// Mitsubishi GX Works2 project: project   PLC: Q03UDV

PROGRAM MAIN
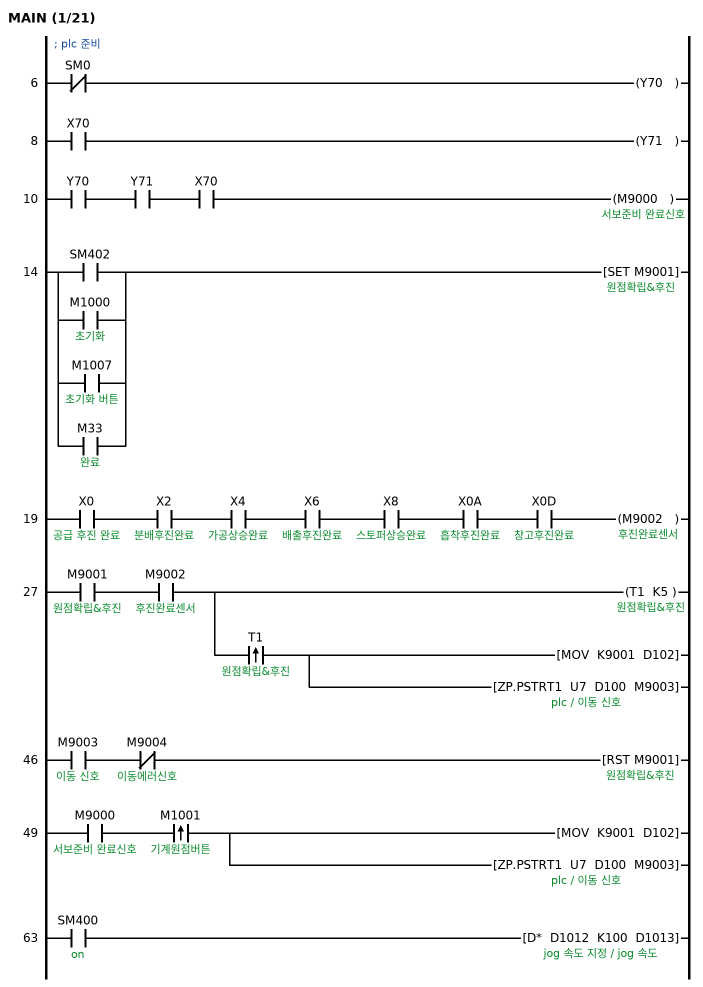
; plc 준비
6     LDI     SM0
      OUT     Y70
8     LD      X70
      OUT     Y71
10    LD      Y70
      AND     Y71
      AND     X70
      OUT     M9000  ; 서보준비 완료신호
14    LD      SM402
      OR      M1000  ; 초기화
      OR      M1007  ; 초기화 버튼
      OR      M33  ; 완료
      SET     M9001  ; 원점확립&후진
19    LD      X0  ; 공급 후진 완료
      AND     X2  ; 분배후진완료
      AND     X4  ; 가공상승완료
      AND     X6  ; 배출후진완료
      AND     X8  ; 스토퍼상승완료
      AND     X0A  ; 흡착후진완료
      AND     X0D  ; 창고후진완료
      OUT     M9002  ; 후진완료센서
27    LD      M9001  ; 원점확립&후진
      AND     M9002  ; 후진완료센서
      OUT     T1 K5  ; 원점확립&후진
      ANDP    T1  ; 원점확립&후진
      MOV     K9001 D102
      ZP.PSTRT1 U7 D100 M9003  ; plc / 이동 신호
46    LD      M9003  ; 이동 신호
      ANI     M9004  ; 이동에러신호
      RST     M9001  ; 원점확립&후진
49    LD      M9000  ; 서보준비 완료신호
      ANDP    M1001  ; 기계원점버튼
      MOV     K9001 D102
      ZP.PSTRT1 U7 D100 M9003
63    LD      SM400  ; on
      D*      D1012 K100 D1013  ; jog 속도 지정 / jog 속도
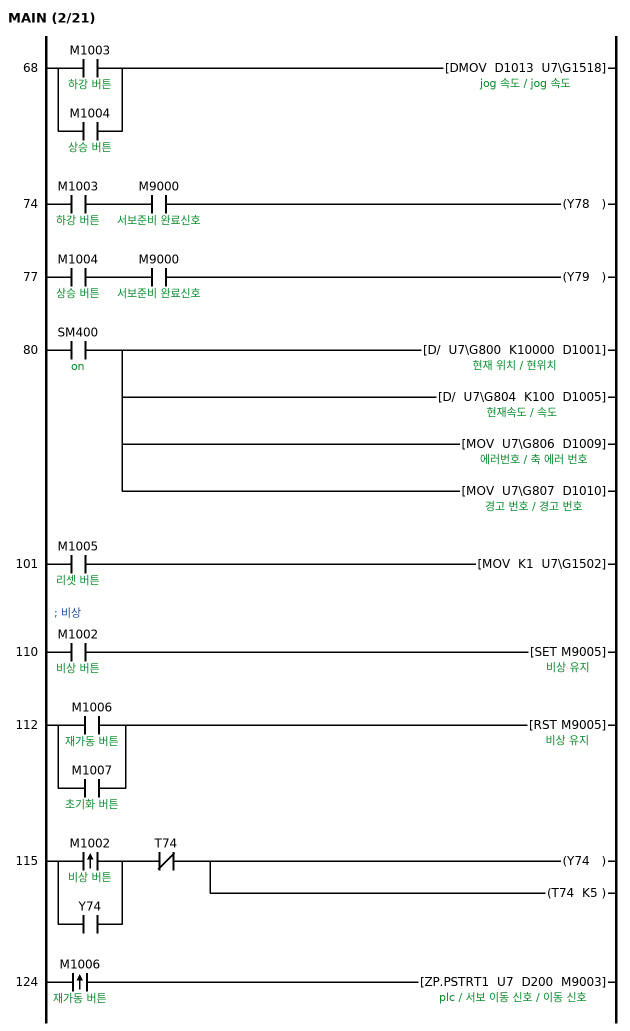
68    LD      M1003  ; 하강 버튼
      OR      M1004  ; 상승 버튼
      DMOV    D1013 U7\G1518  ; jog 속도
74    LD      M1003  ; 하강 버튼
      AND     M9000  ; 서보준비 완료신호
      OUT     Y78
77    LD      M1004  ; 상승 버튼
      AND     M9000  ; 서보준비 완료신호
      OUT     Y79
80    LD      SM400  ; on
      D/      U7\G800 K10000 D1001  ; 현재 위치 / 현위치
      D/      U7\G804 K100 D1005  ; 현재속도 / 속도
      MOV     U7\G806 D1009  ; 에러번호 / 축 에러 번호
      MOV     U7\G807 D1010  ; 경고 번호 / 경고 번호
101   LD      M1005  ; 리셋 버튼
      MOV     K1 U7\G1502
; 비상
110   LD      M1002  ; 비상 버튼
      SET     M9005  ; 비상 유지
112   LD      M1006  ; 재가동 버튼
      OR      M1007  ; 초기화 버튼
      RST     M9005  ; 비상 유지
115   LDP     M1002  ; 비상 버튼
      OR      Y74
      ANI     T74
      OUT     Y74
      OUT     T74 K5
124   LDP     M1006  ; 재가동 버튼
      ZP.PSTRT1 U7 D200 M9003  ; 서보 이동 신호
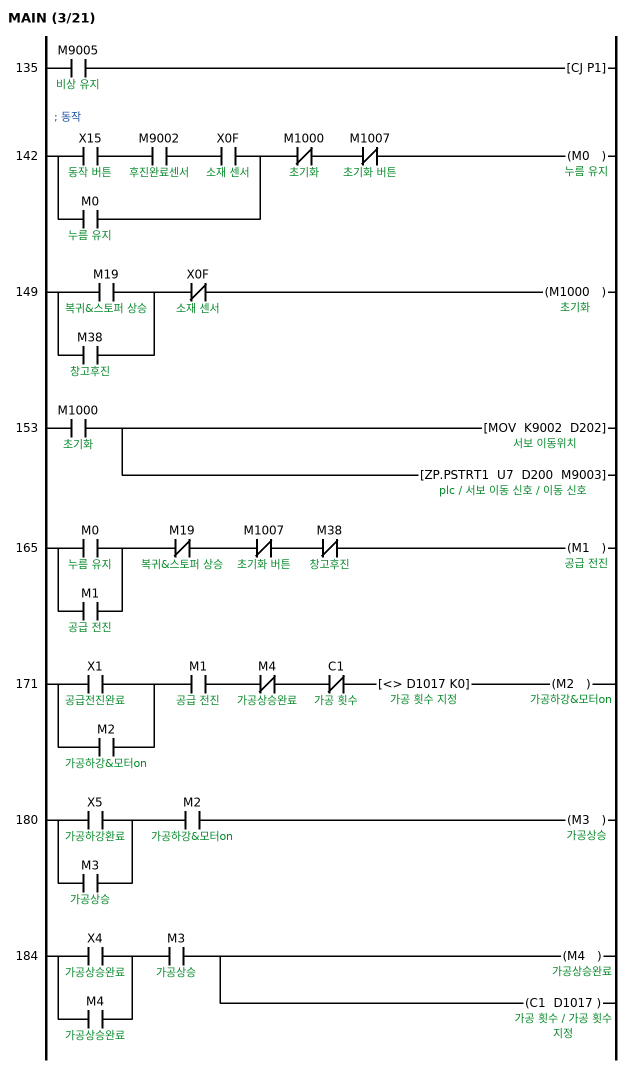
135   LD      M9005  ; 비상 유지
      CJ      P1  ; 비상
; 동작
142   LD      X15  ; 동작 버튼
      AND     M9002  ; 후진완료센서
      AND     X0F  ; 소재 센서
      OR      M0  ; 누름 유지
      ANI     M1000  ; 초기화
      ANI     M1007  ; 초기화 버튼
      OUT     M0  ; 누름 유지
149   LD      M19  ; 복귀&스토퍼 상승
      OR      M38  ; 창고후진
      ANI     X0F  ; 소재 센서
      OUT     M1000  ; 초기화
153   LD      M1000  ; 초기화
      MOV     K9002 D202  ; 서보 이동위치
      ZP.PSTRT1 U7 D200 M9003
165   LD      M0  ; 누름 유지
      OR      M1  ; 공급 전진
      ANI     M19  ; 복귀&스토퍼 상승
      ANI     M1007  ; 초기화 버튼
      ANI     M38  ; 창고후진
      OUT     M1  ; 공급 전진
171   LD      X1  ; 공급전진완료
      OR      M2  ; 가공하강&모터on
      AND     M1  ; 공급 전진
      ANI     M4  ; 가공상승완료
      ANI     C1  ; 가공 횟수
      AND<>   D1017 K0  ; 가공 횟수 지정
      OUT     M2  ; 가공하강&모터on
180   LD      X5  ; 가공하강환료
      OR      M3  ; 가공상승
      AND     M2  ; 가공하강&모터on
      OUT     M3  ; 가공상승
184   LD      X4  ; 가공상승완료
      OR      M4  ; 가공상승완료
      AND     M3  ; 가공상승
      OUT     M4  ; 가공상승완료
      OUT     C1 D1017  ; 가공 횟수 / 가공 횟수 지정
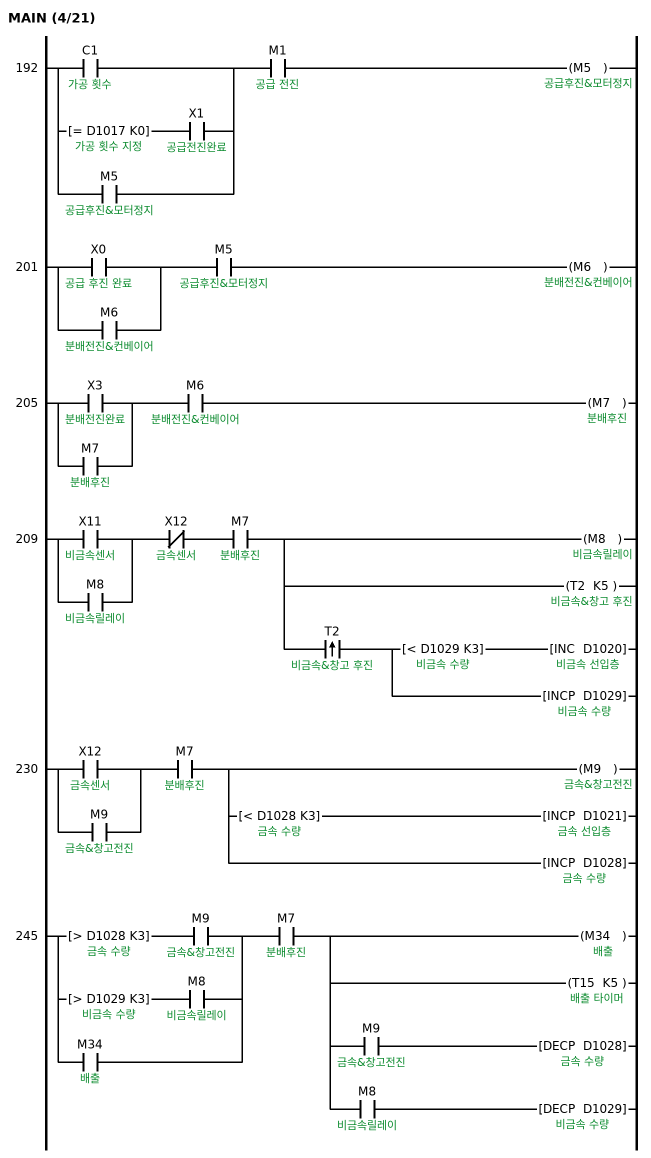
192   LD      C1  ; 가공 횟수
      LD=     D1017 K0  ; 가공 횟수 지정
      AND     X1  ; 공급전진완료
      ORB
      OR      M5  ; 공급후진&모터정지
      AND     M1  ; 공급 전진
      OUT     M5  ; 공급후진&모터정지
201   LD      X0  ; 공급 후진 완료
      OR      M6  ; 분배전진&컨베이어
      AND     M5  ; 공급후진&모터정지
      OUT     M6  ; 분배전진&컨베이어
205   LD      X3  ; 분배전진완료
      OR      M7  ; 분배후진
      AND     M6  ; 분배전진&컨베이어
      OUT     M7  ; 분배후진
209   LD      X11  ; 비금속센서
      OR      M8  ; 비금속릴레이
      ANI     X12  ; 금속센서
      AND     M7  ; 분배후진
      OUT     M8  ; 비금속릴레이
      OUT     T2 K5  ; 비금속&창고 후진
      ANDP    T2  ; 비금속&창고 후진
      MPS
      AND<    D1029 K3  ; 비금속 수량
      INC     D1020  ; 비금속 선입층
      MPP
      INCP    D1029
230   LD      X12  ; 금속센서
      OR      M9  ; 금속&창고전진
      AND     M7  ; 분배후진
      OUT     M9  ; 금속&창고전진
      MPS
      AND<    D1028 K3  ; 금속 수량
      INCP    D1021  ; 금속 선입층
      MPP
      INCP    D1028
245   LD>     D1028 K3  ; 금속 수량
      AND     M9  ; 금속&창고전진
      LD>     D1029 K3  ; 비금속 수량
      AND     M8  ; 비금속릴레이
      ORB
      OR      M34  ; 배출
      AND     M7  ; 분배후진
      OUT     M34  ; 배출
      OUT     T15 K5  ; 배출 타이머
      MPS
      AND     M9  ; 금속&창고전진
      DECP    D1028
      MPP
      AND     M8  ; 비금속릴레이
      DECP    D1029
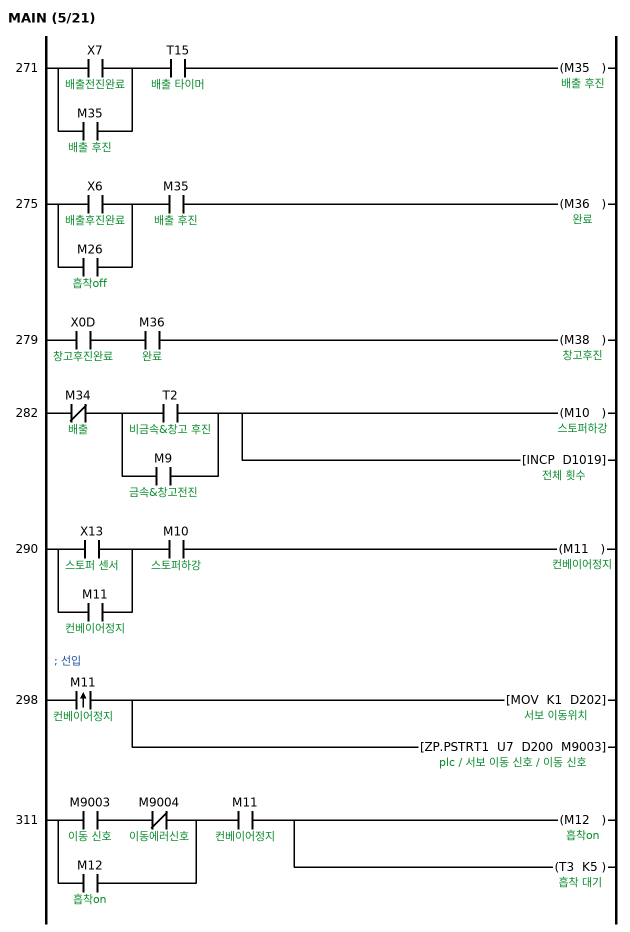
271   LD      X7  ; 배출전진완료
      OR      M35  ; 배출 후진
      AND     T15  ; 배출 타이머
      OUT     M35  ; 배출 후진
275   LD      X6  ; 배출후진완료
      OR      M26  ; 흡착off
      AND     M35  ; 배출 후진
      OUT     M36  ; 완료
279   LD      X0D  ; 창고후진완료
      AND     M36  ; 완료
      OUT     M38  ; 창고후진
282   LDI     M34  ; 배출
      LD      T2  ; 비금속&창고 후진
      OR      M9  ; 금속&창고전진
      ANB
      OUT     M10  ; 스토퍼하강
      INCP    D1019  ; 전체 횟수
290   LD      X13  ; 스토퍼 센서
      OR      M11  ; 컨베이어정지
      AND     M10  ; 스토퍼하강
      OUT     M11  ; 컨베이어정지
; 선입
298   LDP     M11  ; 컨베이어정지
      MOV     K1 D202
      ZP.PSTRT1 U7 D200 M9003
311   LD      M9003  ; 이동 신호
      ANI     M9004  ; 이동에러신호
      OR      M12  ; 흡착on
      AND     M11  ; 컨베이어정지
      OUT     M12  ; 흡착on
      OUT     T3 K5  ; 흡착 대기
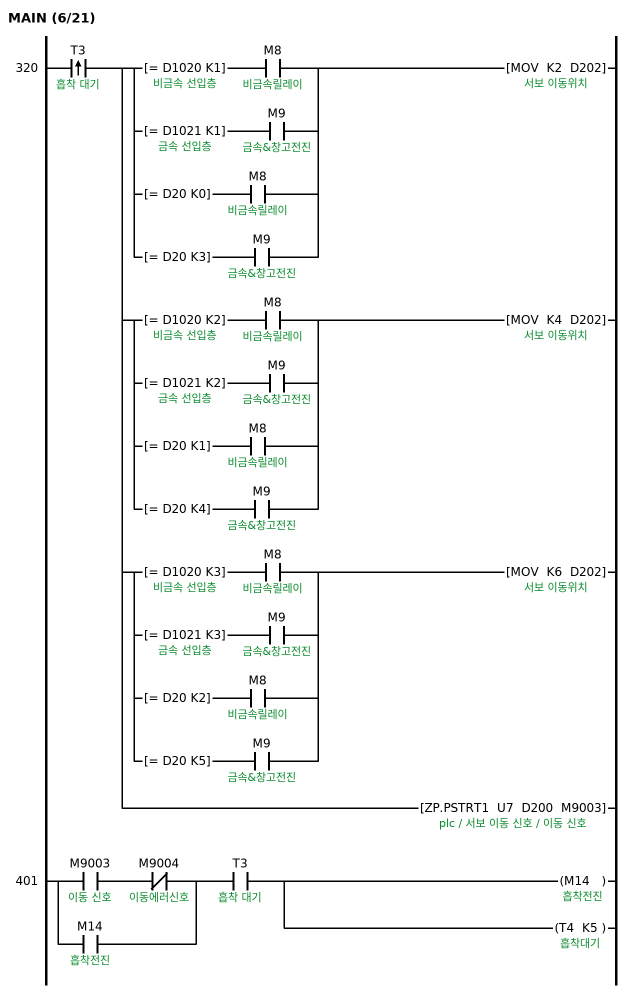
320   LDP     T3  ; 흡착 대기
      MPS
      LD=     D1020 K1  ; 비금속 선입층
      AND     M8  ; 비금속릴레이
      LD=     D1021 K1  ; 금속 선입층
      AND     M9  ; 금속&창고전진
      ORB
      LD=     D20 K0
      AND     M8  ; 비금속릴레이
      ORB
      LD=     D20 K3
      AND     M9  ; 금속&창고전진
      ORB
      ANB
      MOV     K2 D202
      MRD
      LD=     D1020 K2  ; 비금속 선입층
      AND     M8  ; 비금속릴레이
      LD=     D1021 K2  ; 금속 선입층
      AND     M9  ; 금속&창고전진
      ORB
      LD=     D20 K1
      AND     M8  ; 비금속릴레이
      ORB
      LD=     D20 K4
      AND     M9  ; 금속&창고전진
      ORB
      ANB
      MOV     K4 D202
      MRD
      LD=     D1020 K3  ; 비금속 선입층
      AND     M8  ; 비금속릴레이
      LD=     D1021 K3  ; 금속 선입층
      AND     M9  ; 금속&창고전진
      ORB
      LD=     D20 K2
      AND     M8  ; 비금속릴레이
      ORB
      LD=     D20 K5
      AND     M9  ; 금속&창고전진
      ORB
      ANB
      MOV     K6 D202
      MPP
      ZP.PSTRT1 U7 D200 M9003
401   LD      M9003  ; 이동 신호
      ANI     M9004  ; 이동에러신호
      OR      M14  ; 흡착전진
      AND     T3  ; 흡착 대기
      OUT     M14  ; 흡착전진
      OUT     T4 K5  ; 흡착대기
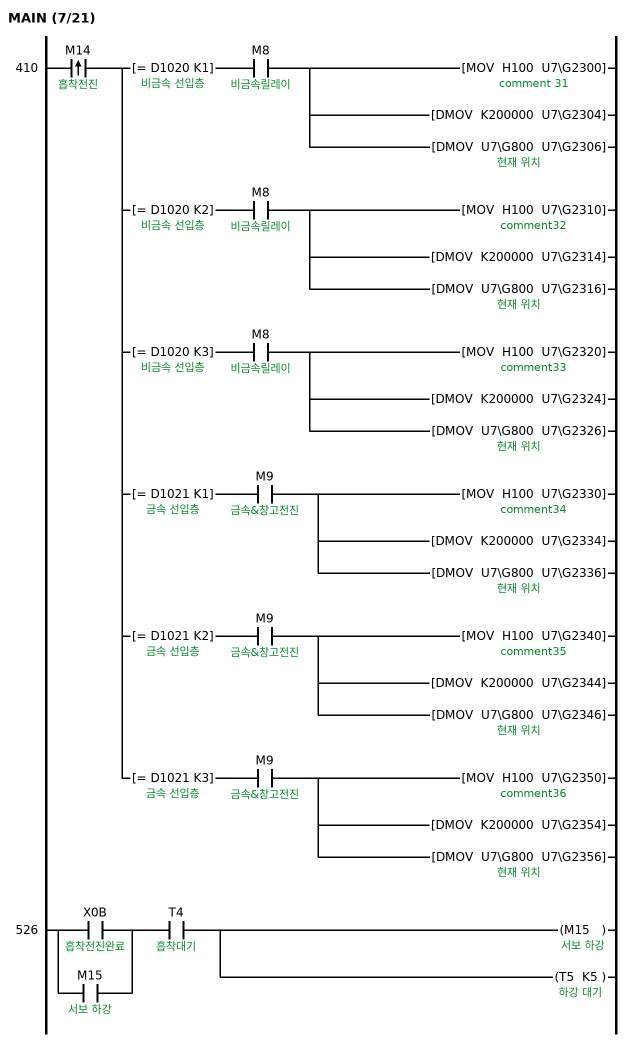
410   LDP     M14  ; 흡착전진
      MPS
      AND=    D1020 K1  ; 비금속 선입층
      AND     M8  ; 비금속릴레이
      MOV     H100 U7\G2300  ; comment 31
      DMOV    K200000 U7\G2304
      DMOV    U7\G800 U7\G2306
      MRD
      AND=    D1020 K2  ; 비금속 선입층
      AND     M8  ; 비금속릴레이
      MOV     H100 U7\G2310  ; comment32
      DMOV    K200000 U7\G2314
      DMOV    U7\G800 U7\G2316
      MRD
      AND=    D1020 K3  ; 비금속 선입층
      AND     M8  ; 비금속릴레이
      MOV     H100 U7\G2320  ; comment33
      DMOV    K200000 U7\G2324
      DMOV    U7\G800 U7\G2326
      MRD
      AND=    D1021 K1  ; 금속 선입층
      AND     M9  ; 금속&창고전진
      MOV     H100 U7\G2330  ; comment34
      DMOV    K200000 U7\G2334
      DMOV    U7\G800 U7\G2336
      MRD
      AND=    D1021 K2  ; 금속 선입층
      AND     M9  ; 금속&창고전진
      MOV     H100 U7\G2340  ; comment35
      DMOV    K200000 U7\G2344
      DMOV    U7\G800 U7\G2346
      MPP
      AND=    D1021 K3  ; 금속 선입층
      AND     M9  ; 금속&창고전진
      MOV     H100 U7\G2350  ; comment36
      DMOV    K200000 U7\G2354
      DMOV    U7\G800 U7\G2356
526   LD      X0B  ; 흡착전진완료
      OR      M15  ; 서보 하강
      AND     T4  ; 흡착대기
      OUT     M15  ; 서보 하강
      OUT     T5 K5  ; 하강 대기
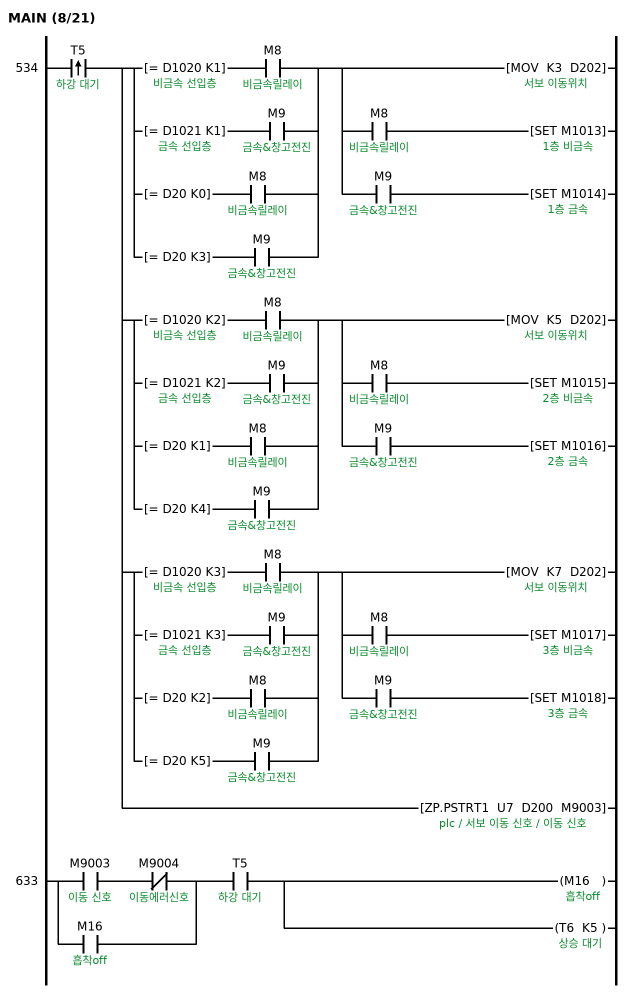
534   LDP     T5  ; 하강 대기
      MPS
      LD=     D1020 K1  ; 비금속 선입층
      AND     M8  ; 비금속릴레이
      LD=     D1021 K1  ; 금속 선입층
      AND     M9  ; 금속&창고전진
      ORB
      LD=     D20 K0
      AND     M8  ; 비금속릴레이
      ORB
      LD=     D20 K3
      AND     M9  ; 금속&창고전진
      ORB
      ANB
      MOV     K3 D202
      MPS
      AND     M8  ; 비금속릴레이
      SET     M1013  ; 1층 비금속
      MPP
      AND     M9  ; 금속&창고전진
      SET     M1014  ; 1층 금속
      MRD
      LD=     D1020 K2  ; 비금속 선입층
      AND     M8  ; 비금속릴레이
      LD=     D1021 K2  ; 금속 선입층
      AND     M9  ; 금속&창고전진
      ORB
      LD=     D20 K1
      AND     M8  ; 비금속릴레이
      ORB
      LD=     D20 K4
      AND     M9  ; 금속&창고전진
      ORB
      ANB
      MOV     K5 D202
      MPS
      AND     M8  ; 비금속릴레이
      SET     M1015  ; 2층 비금속
      MPP
      AND     M9  ; 금속&창고전진
      SET     M1016  ; 2층 금속
      MRD
      LD=     D1020 K3  ; 비금속 선입층
      AND     M8  ; 비금속릴레이
      LD=     D1021 K3  ; 금속 선입층
      AND     M9  ; 금속&창고전진
      ORB
      LD=     D20 K2
      AND     M8  ; 비금속릴레이
      ORB
      LD=     D20 K5
      AND     M9  ; 금속&창고전진
      ORB
      ANB
      MOV     K7 D202
      MPS
      AND     M8  ; 비금속릴레이
      SET     M1017  ; 3층 비금속
      MPP
      AND     M9  ; 금속&창고전진
      SET     M1018  ; 3층 금속
      MPP
      ZP.PSTRT1 U7 D200 M9003
633   LD      M9003  ; 이동 신호
      ANI     M9004  ; 이동에러신호
      OR      M16  ; 흡착off
      AND     T5  ; 하강 대기
      OUT     M16  ; 흡착off
      OUT     T6 K5  ; 상승 대기
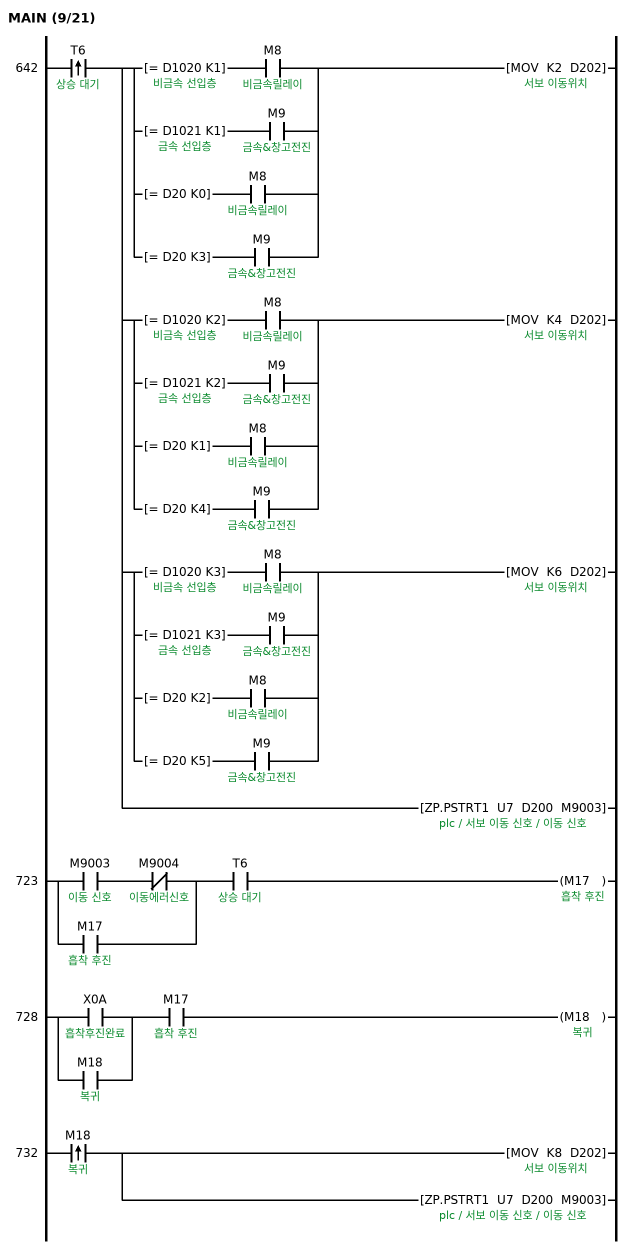
642   LDP     T6  ; 상승 대기
      MPS
      LD=     D1020 K1  ; 비금속 선입층
      AND     M8  ; 비금속릴레이
      LD=     D1021 K1  ; 금속 선입층
      AND     M9  ; 금속&창고전진
      ORB
      LD=     D20 K0
      AND     M8  ; 비금속릴레이
      ORB
      LD=     D20 K3
      AND     M9  ; 금속&창고전진
      ORB
      ANB
      MOV     K2 D202
      MRD
      LD=     D1020 K2  ; 비금속 선입층
      AND     M8  ; 비금속릴레이
      LD=     D1021 K2  ; 금속 선입층
      AND     M9  ; 금속&창고전진
      ORB
      LD=     D20 K1
      AND     M8  ; 비금속릴레이
      ORB
      LD=     D20 K4
      AND     M9  ; 금속&창고전진
      ORB
      ANB
      MOV     K4 D202
      MRD
      LD=     D1020 K3  ; 비금속 선입층
      AND     M8  ; 비금속릴레이
      LD=     D1021 K3  ; 금속 선입층
      AND     M9  ; 금속&창고전진
      ORB
      LD=     D20 K2
      AND     M8  ; 비금속릴레이
      ORB
      LD=     D20 K5
      AND     M9  ; 금속&창고전진
      ORB
      ANB
      MOV     K6 D202
      MPP
      ZP.PSTRT1 U7 D200 M9003
723   LD      M9003  ; 이동 신호
      ANI     M9004  ; 이동에러신호
      OR      M17  ; 흡착 후진
      AND     T6  ; 상승 대기
      OUT     M17  ; 흡착 후진
728   LD      X0A  ; 흡착후진완료
      OR      M18  ; 복귀
      AND     M17  ; 흡착 후진
      OUT     M18  ; 복귀
732   LDP     M18  ; 복귀
      MOV     K8 D202
      ZP.PSTRT1 U7 D200 M9003
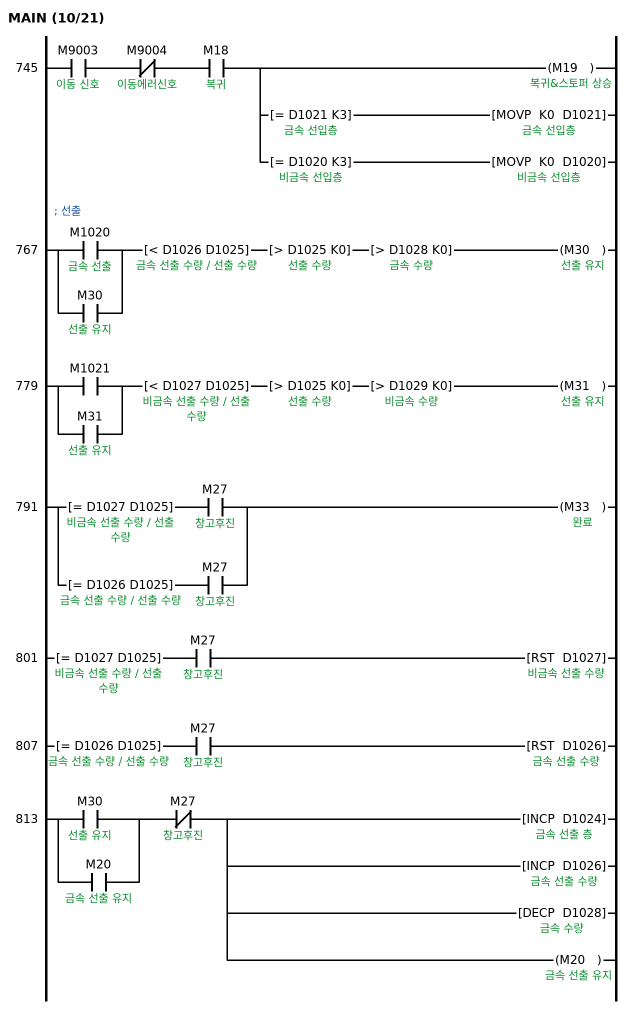
745   LD      M9003  ; 이동 신호
      ANI     M9004  ; 이동에러신호
      AND     M18  ; 복귀
      OUT     M19  ; 복귀&스토퍼 상승
      MPS
      AND=    D1021 K3  ; 금속 선입층
      MOVP    K0 D1021
      MPP
      AND=    D1020 K3  ; 비금속 선입층
      MOVP    K0 D1020
; 선출
767   LD      M1020  ; 금속 선출
      OR      M30  ; 선출 유지
      AND<    D1026 D1025  ; 금속 선출 수량 / 선출 수량
      AND>    D1025 K0  ; 선출 수량
      AND>    D1028 K0  ; 금속 수량
      OUT     M30  ; 선출 유지
779   LD      M1021
      OR      M31  ; 선출 유지
      AND<    D1027 D1025  ; 비금속 선출 수량 / 선출 수량
      AND>    D1025 K0  ; 선출 수량
      AND>    D1029 K0  ; 비금속 수량
      OUT     M31  ; 선출 유지
791   LD=     D1027 D1025  ; 비금속 선출 수량 / 선출 수량
      AND     M27  ; 창고후진
      LD=     D1026 D1025  ; 금속 선출 수량 / 선출 수량
      AND     M27  ; 창고후진
      ORB
      OUT     M33  ; 완료
801   LD=     D1027 D1025  ; 비금속 선출 수량 / 선출 수량
      AND     M27  ; 창고후진
      RST     D1027  ; 비금속 선출 수량
807   LD=     D1026 D1025  ; 금속 선출 수량 / 선출 수량
      AND     M27  ; 창고후진
      RST     D1026  ; 금속 선출 수량
813   LD      M30  ; 선출 유지
      OR      M20  ; 금속 선출 유지
      ANI     M27  ; 창고후진
      INCP    D1024  ; 금속 선출 층
      INCP    D1026
      DECP    D1028
      OUT     M20  ; 금속 선출 유지
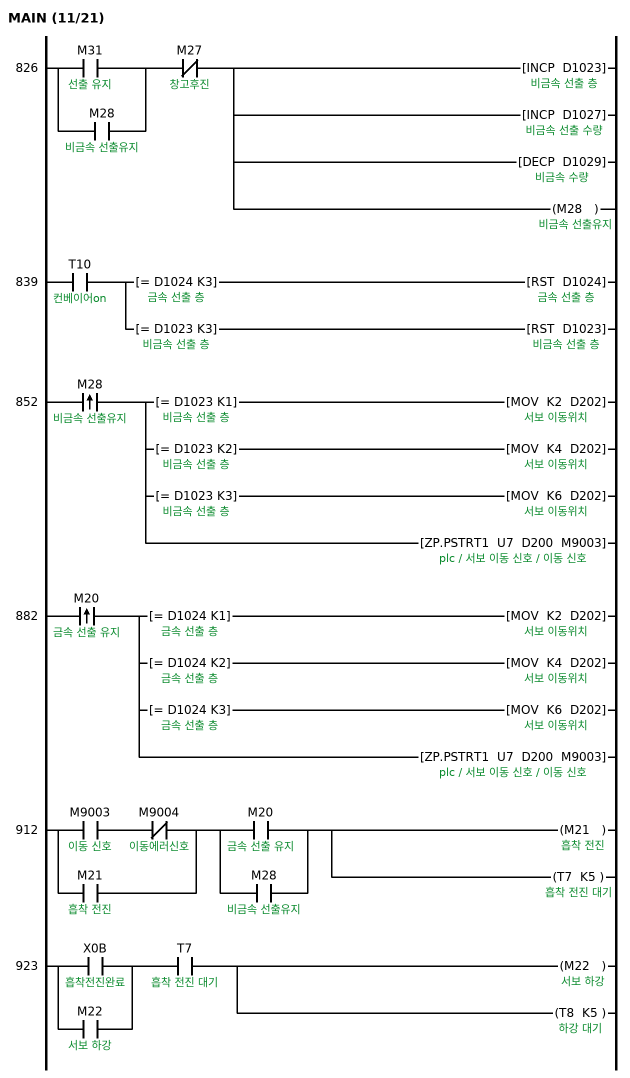
826   LD      M31  ; 선출 유지
      OR      M28  ; 비금속 선출유지
      ANI     M27  ; 창고후진
      INCP    D1023  ; 비금속 선출 층
      INCP    D1027
      DECP    D1029
      OUT     M28  ; 비금속 선출유지
839   LD      T10  ; 컨베이어on
      MPS
      AND=    D1024 K3  ; 금속 선출 층
      RST     D1024  ; 금속 선출 층
      MPP
      AND=    D1023 K3  ; 비금속 선출 층
      RST     D1023  ; 비금속 선출 층
852   LDP     M28  ; 비금속 선출유지
      MPS
      AND=    D1023 K1  ; 비금속 선출 층
      MOV     K2 D202
      MRD
      AND=    D1023 K2  ; 비금속 선출 층
      MOV     K4 D202
      MRD
      AND=    D1023 K3  ; 비금속 선출 층
      MOV     K6 D202
      MPP
      ZP.PSTRT1 U7 D200 M9003
882   LDP     M20  ; 금속 선출 유지
      MPS
      AND=    D1024 K1  ; 금속 선출 층
      MOV     K2 D202
      MRD
      AND=    D1024 K2  ; 금속 선출 층
      MOV     K4 D202
      MRD
      AND=    D1024 K3  ; 금속 선출 층
      MOV     K6 D202
      MPP
      ZP.PSTRT1 U7 D200 M9003
912   LD      M9003  ; 이동 신호
      ANI     M9004  ; 이동에러신호
      OR      M21  ; 흡착 전진
      LD      M20  ; 금속 선출 유지
      OR      M28  ; 비금속 선출유지
      ANB
      OUT     M21  ; 흡착 전진
      OUT     T7 K5  ; 흡착 전진 대기
923   LD      X0B  ; 흡착전진완료
      OR      M22  ; 서보 하강
      AND     T7  ; 흡착 전진 대기
      OUT     M22  ; 서보 하강
      OUT     T8 K5  ; 하강 대기
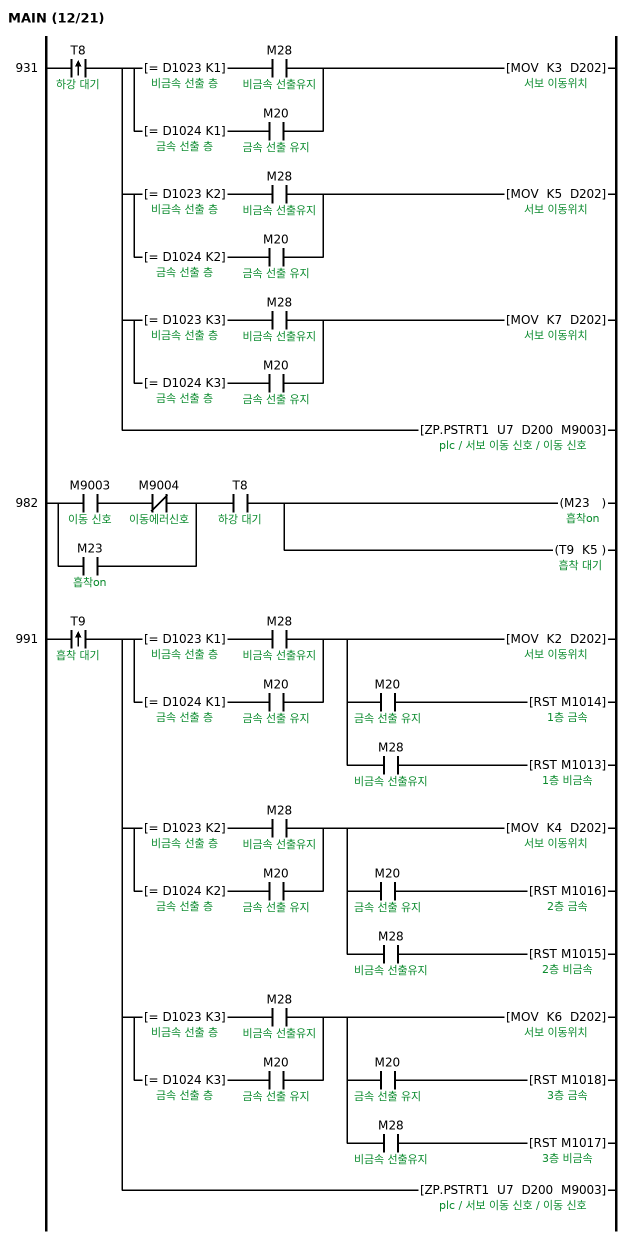
931   LDP     T8  ; 하강 대기
      MPS
      LD=     D1023 K1  ; 비금속 선출 층
      AND     M28  ; 비금속 선출유지
      LD=     D1024 K1  ; 금속 선출 층
      AND     M20  ; 금속 선출 유지
      ORB
      ANB
      MOV     K3 D202
      MRD
      LD=     D1023 K2  ; 비금속 선출 층
      AND     M28  ; 비금속 선출유지
      LD=     D1024 K2  ; 금속 선출 층
      AND     M20  ; 금속 선출 유지
      ORB
      ANB
      MOV     K5 D202
      MRD
      LD=     D1023 K3  ; 비금속 선출 층
      AND     M28  ; 비금속 선출유지
      LD=     D1024 K3  ; 금속 선출 층
      AND     M20  ; 금속 선출 유지
      ORB
      ANB
      MOV     K7 D202
      MPP
      ZP.PSTRT1 U7 D200 M9003
982   LD      M9003  ; 이동 신호
      ANI     M9004  ; 이동에러신호
      OR      M23  ; 흡착on
      AND     T8  ; 하강 대기
      OUT     M23  ; 흡착on
      OUT     T9 K5  ; 흡착 대기
991   LDP     T9  ; 흡착 대기
      MPS
      LD=     D1023 K1  ; 비금속 선출 층
      AND     M28  ; 비금속 선출유지
      LD=     D1024 K1  ; 금속 선출 층
      AND     M20  ; 금속 선출 유지
      ORB
      ANB
      MOV     K2 D202
      MPS
      AND     M20  ; 금속 선출 유지
      RST     M1014  ; 1층 금속
      MPP
      AND     M28  ; 비금속 선출유지
      RST     M1013  ; 1층 비금속
      MRD
      LD=     D1023 K2  ; 비금속 선출 층
      AND     M28  ; 비금속 선출유지
      LD=     D1024 K2  ; 금속 선출 층
      AND     M20  ; 금속 선출 유지
      ORB
      ANB
      MOV     K4 D202
      MPS
      AND     M20  ; 금속 선출 유지
      RST     M1016  ; 2층 금속
      MPP
      AND     M28  ; 비금속 선출유지
      RST     M1015  ; 2층 비금속
      MRD
      LD=     D1023 K3  ; 비금속 선출 층
      AND     M28  ; 비금속 선출유지
      LD=     D1024 K3  ; 금속 선출 층
      AND     M20  ; 금속 선출 유지
      ORB
      ANB
      MOV     K6 D202
      MPS
      AND     M20  ; 금속 선출 유지
      RST     M1018  ; 3층 금속
      MPP
      AND     M28  ; 비금속 선출유지
      RST     M1017  ; 3층 비금속
      MPP
      ZP.PSTRT1 U7 D200 M9003
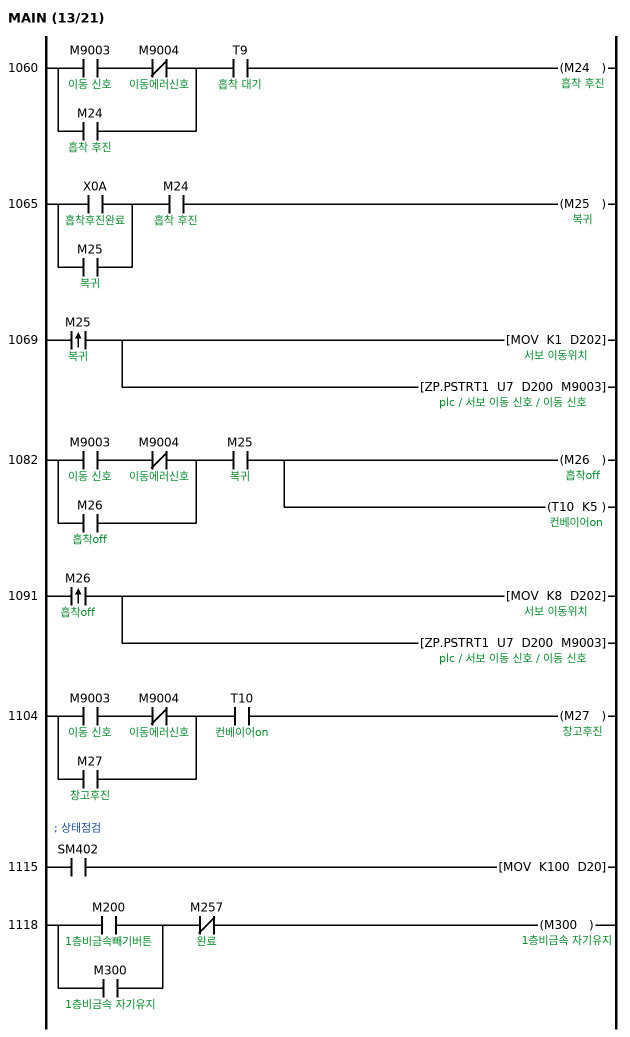
1060  LD      M9003  ; 이동 신호
      ANI     M9004  ; 이동에러신호
      OR      M24  ; 흡착 후진
      AND     T9  ; 흡착 대기
      OUT     M24  ; 흡착 후진
1065  LD      X0A  ; 흡착후진완료
      OR      M25  ; 복귀
      AND     M24  ; 흡착 후진
      OUT     M25  ; 복귀
1069  LDP     M25  ; 복귀
      MOV     K1 D202
      ZP.PSTRT1 U7 D200 M9003
1082  LD      M9003  ; 이동 신호
      ANI     M9004  ; 이동에러신호
      OR      M26  ; 흡착off
      AND     M25  ; 복귀
      OUT     M26  ; 흡착off
      OUT     T10 K5  ; 컨베이어on
1091  LDP     M26  ; 흡착off
      MOV     K8 D202
      ZP.PSTRT1 U7 D200 M9003
1104  LD      M9003  ; 이동 신호
      ANI     M9004  ; 이동에러신호
      OR      M27  ; 창고후진
      AND     T10  ; 컨베이어on
      OUT     M27  ; 창고후진
; 상태점검
1115  LD      SM402
      MOV     K100 D20
1118  LD      M200  ; 1층비금속빼기버튼
      OR      M300  ; 1층비금속 자기유지
      ANI     M257  ; 완료
      OUT     M300  ; 1층비금속 자기유지
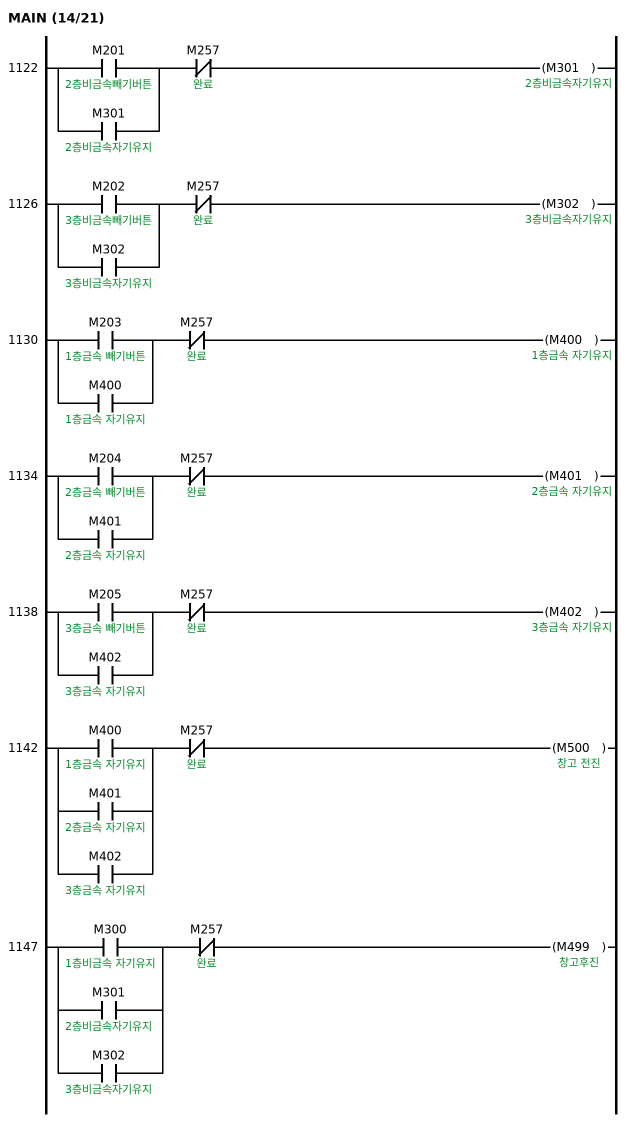
1122  LD      M201  ; 2층비금속빼기버튼
      OR      M301  ; 2층비금속자기유지
      ANI     M257  ; 완료
      OUT     M301  ; 2층비금속자기유지
1126  LD      M202  ; 3층비금속빼기버튼
      OR      M302  ; 3층비금속자기유지
      ANI     M257  ; 완료
      OUT     M302  ; 3층비금속자기유지
1130  LD      M203  ; 1층금속 빼기버튼
      OR      M400  ; 1층금속 자기유지
      ANI     M257  ; 완료
      OUT     M400  ; 1층금속 자기유지
1134  LD      M204  ; 2층금속 빼기버튼
      OR      M401  ; 2층금속 자기유지
      ANI     M257  ; 완료
      OUT     M401  ; 2층금속 자기유지
1138  LD      M205  ; 3층금속 빼기버튼
      OR      M402  ; 3층금속 자기유지
      ANI     M257  ; 완료
      OUT     M402  ; 3층금속 자기유지
1142  LD      M400  ; 1층금속 자기유지
      OR      M401  ; 2층금속 자기유지
      OR      M402  ; 3층금속 자기유지
      ANI     M257  ; 완료
      OUT     M500  ; 창고 전진
1147  LD      M300  ; 1층비금속 자기유지
      OR      M301  ; 2층비금속자기유지
      OR      M302  ; 3층비금속자기유지
      ANI     M257  ; 완료
      OUT     M499  ; 창고후진
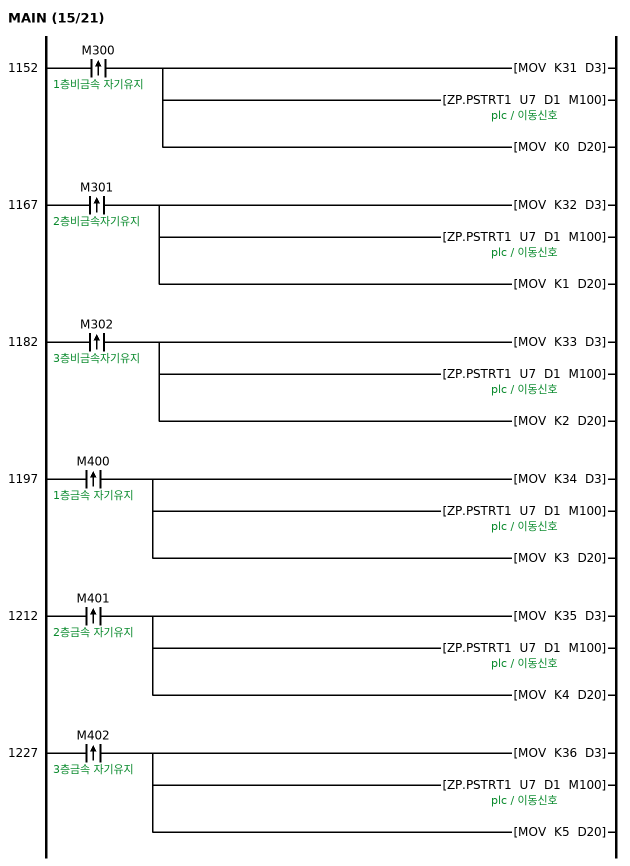
1152  LDP     M300  ; 1층비금속 자기유지
      MOV     K31 D3
      ZP.PSTRT1 U7 D1 M100  ; 이동신호
      MOV     K0 D20
1167  LDP     M301  ; 2층비금속자기유지
      MOV     K32 D3
      ZP.PSTRT1 U7 D1 M100
      MOV     K1 D20
1182  LDP     M302  ; 3층비금속자기유지
      MOV     K33 D3
      ZP.PSTRT1 U7 D1 M100
      MOV     K2 D20
1197  LDP     M400  ; 1층금속 자기유지
      MOV     K34 D3
      ZP.PSTRT1 U7 D1 M100
      MOV     K3 D20
1212  LDP     M401  ; 2층금속 자기유지
      MOV     K35 D3
      ZP.PSTRT1 U7 D1 M100
      MOV     K4 D20
1227  LDP     M402  ; 3층금속 자기유지
      MOV     K36 D3
      ZP.PSTRT1 U7 D1 M100
      MOV     K5 D20
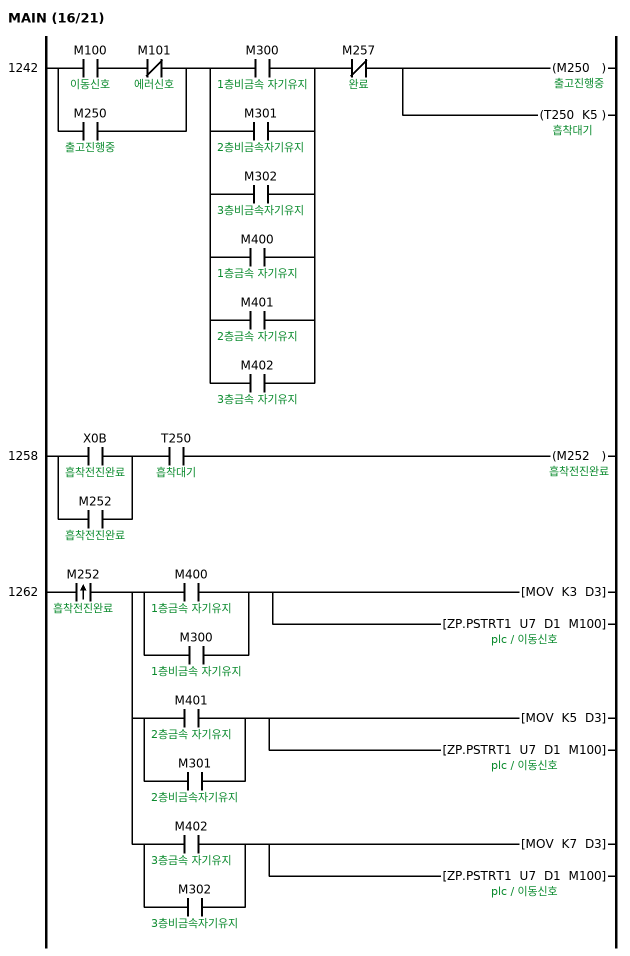
1242  LD      M100  ; 이동신호
      ANI     M101  ; 에러신호
      OR      M250  ; 출고진행중
      LD      M300  ; 1층비금속 자기유지
      OR      M301  ; 2층비금속자기유지
      OR      M302  ; 3층비금속자기유지
      OR      M400  ; 1층금속 자기유지
      OR      M401  ; 2층금속 자기유지
      OR      M402  ; 3층금속 자기유지
      ANB
      ANI     M257  ; 완료
      OUT     M250  ; 출고진행중
      OUT     T250 K5  ; 흡착대기
1258  LD      X0B  ; 흡착전진완료
      OR      M252  ; 흡착전진완료
      AND     T250  ; 흡착대기
      OUT     M252  ; 흡착전진완료
1262  LDP     M252  ; 흡착전진완료
      MPS
      LD      M400  ; 1층금속 자기유지
      OR      M300  ; 1층비금속 자기유지
      ANB
      MOV     K3 D3
      ZP.PSTRT1 U7 D1 M100
      MRD
      LD      M401  ; 2층금속 자기유지
      OR      M301  ; 2층비금속자기유지
      ANB
      MOV     K5 D3
      ZP.PSTRT1 U7 D1 M100
      MPP
      LD      M402  ; 3층금속 자기유지
      OR      M302  ; 3층비금속자기유지
      ANB
      MOV     K7 D3
      ZP.PSTRT1 U7 D1 M100
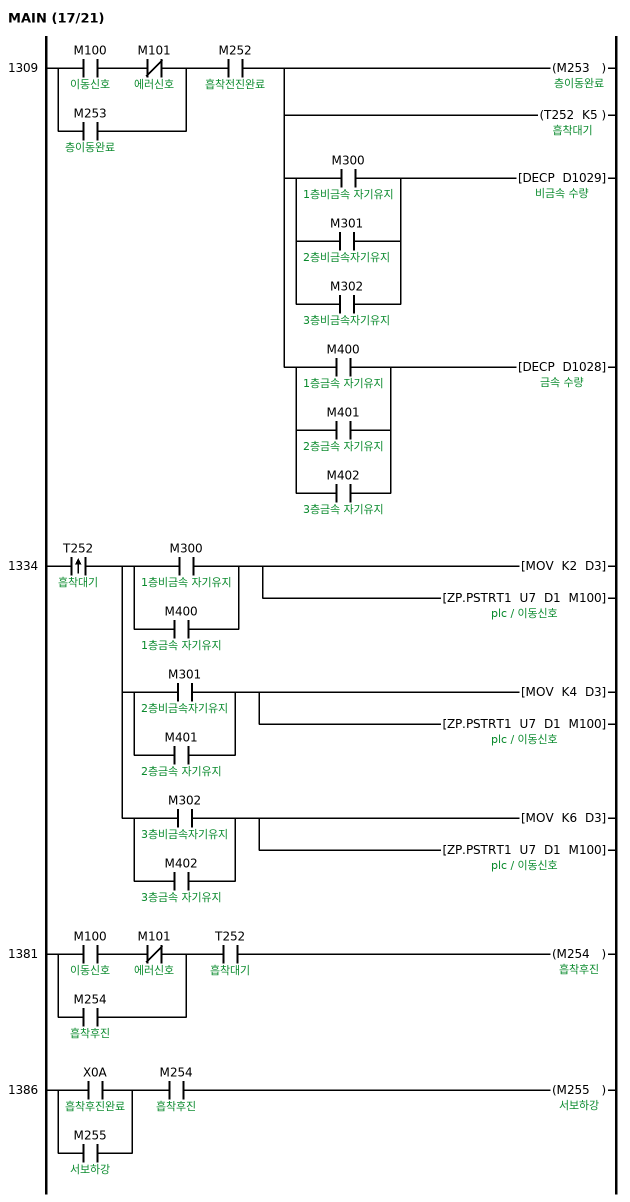
1309  LD      M100  ; 이동신호
      ANI     M101  ; 에러신호
      OR      M253  ; 층이동완료
      AND     M252  ; 흡착전진완료
      OUT     M253  ; 층이동완료
      OUT     T252 K5  ; 흡착대기
      MPS
      LD      M300  ; 1층비금속 자기유지
      OR      M301  ; 2층비금속자기유지
      OR      M302  ; 3층비금속자기유지
      ANB
      DECP    D1029
      MPP
      LD      M400  ; 1층금속 자기유지
      OR      M401  ; 2층금속 자기유지
      OR      M402  ; 3층금속 자기유지
      ANB
      DECP    D1028
1334  LDP     T252  ; 흡착대기
      MPS
      LD      M300  ; 1층비금속 자기유지
      OR      M400  ; 1층금속 자기유지
      ANB
      MOV     K2 D3
      ZP.PSTRT1 U7 D1 M100
      MRD
      LD      M301  ; 2층비금속자기유지
      OR      M401  ; 2층금속 자기유지
      ANB
      MOV     K4 D3
      ZP.PSTRT1 U7 D1 M100
      MPP
      LD      M302  ; 3층비금속자기유지
      OR      M402  ; 3층금속 자기유지
      ANB
      MOV     K6 D3
      ZP.PSTRT1 U7 D1 M100
1381  LD      M100  ; 이동신호
      ANI     M101  ; 에러신호
      OR      M254  ; 흡착후진
      AND     T252  ; 흡착대기
      OUT     M254  ; 흡착후진
1386  LD      X0A  ; 흡착후진완료
      OR      M255  ; 서보하강
      AND     M254  ; 흡착후진
      OUT     M255  ; 서보하강
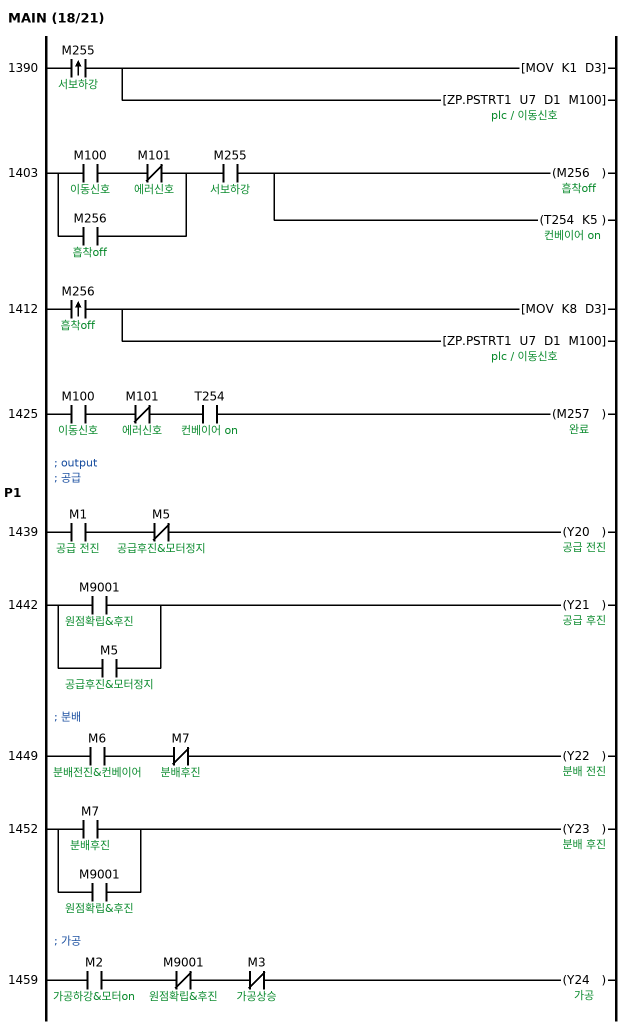
1390  LDP     M255  ; 서보하강
      MOV     K1 D3
      ZP.PSTRT1 U7 D1 M100
1403  LD      M100  ; 이동신호
      ANI     M101  ; 에러신호
      OR      M256  ; 흡착off
      AND     M255  ; 서보하강
      OUT     M256  ; 흡착off
      OUT     T254 K5  ; 컨베이어 on
1412  LDP     M256  ; 흡착off
      MOV     K8 D3
      ZP.PSTRT1 U7 D1 M100
1425  LD      M100  ; 이동신호
      ANI     M101  ; 에러신호
      AND     T254  ; 컨베이어 on
      OUT     M257  ; 완료
; output
; 공급
      P1
1439  LD      M1  ; 공급 전진
      ANI     M5  ; 공급후진&모터정지
      OUT     Y20  ; 공급 전진
1442  LD      M9001  ; 원점확립&후진
      OR      M5  ; 공급후진&모터정지
      OUT     Y21  ; 공급 후진
; 분배
1449  LD      M6  ; 분배전진&컨베이어
      ANI     M7  ; 분배후진
      OUT     Y22  ; 분배 전진
1452  LD      M7  ; 분배후진
      OR      M9001  ; 원점확립&후진
      OUT     Y23  ; 분배 후진
; 가공
1459  LD      M2  ; 가공하강&모터on
      ANI     M9001  ; 원점확립&후진
      ANI     M3  ; 가공상승
      OUT     Y24  ; 가공
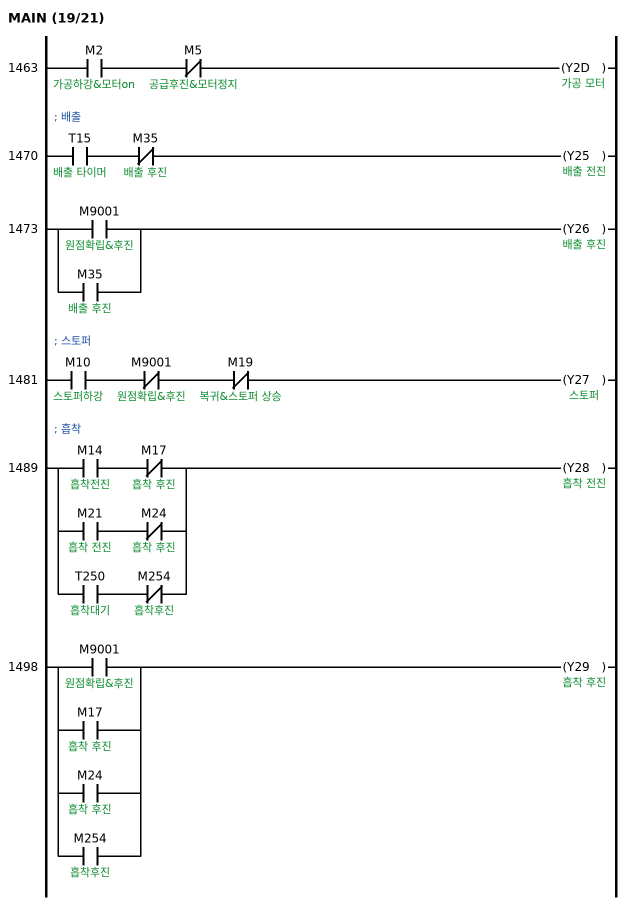
1463  LD      M2  ; 가공하강&모터on
      ANI     M5  ; 공급후진&모터정지
      OUT     Y2D  ; 가공 모터
; 배출
1470  LD      T15  ; 배출 타이머
      ANI     M35  ; 배출 후진
      OUT     Y25  ; 배출 전진
1473  LD      M9001  ; 원점확립&후진
      OR      M35  ; 배출 후진
      OUT     Y26  ; 배출 후진
; 스토퍼
1481  LD      M10  ; 스토퍼하강
      ANI     M9001  ; 원점확립&후진
      ANI     M19  ; 복귀&스토퍼 상승
      OUT     Y27  ; 스토퍼
; 흡착
1489  LD      M14  ; 흡착전진
      ANI     M17  ; 흡착 후진
      LD      M21  ; 흡착 전진
      ANI     M24  ; 흡착 후진
      ORB
      LD      T250  ; 흡착대기
      ANI     M254  ; 흡착후진
      ORB
      OUT     Y28  ; 흡착 전진
1498  LD      M9001  ; 원점확립&후진
      OR      M17  ; 흡착 후진
      OR      M24  ; 흡착 후진
      OR      M254  ; 흡착후진
      OUT     Y29  ; 흡착 후진
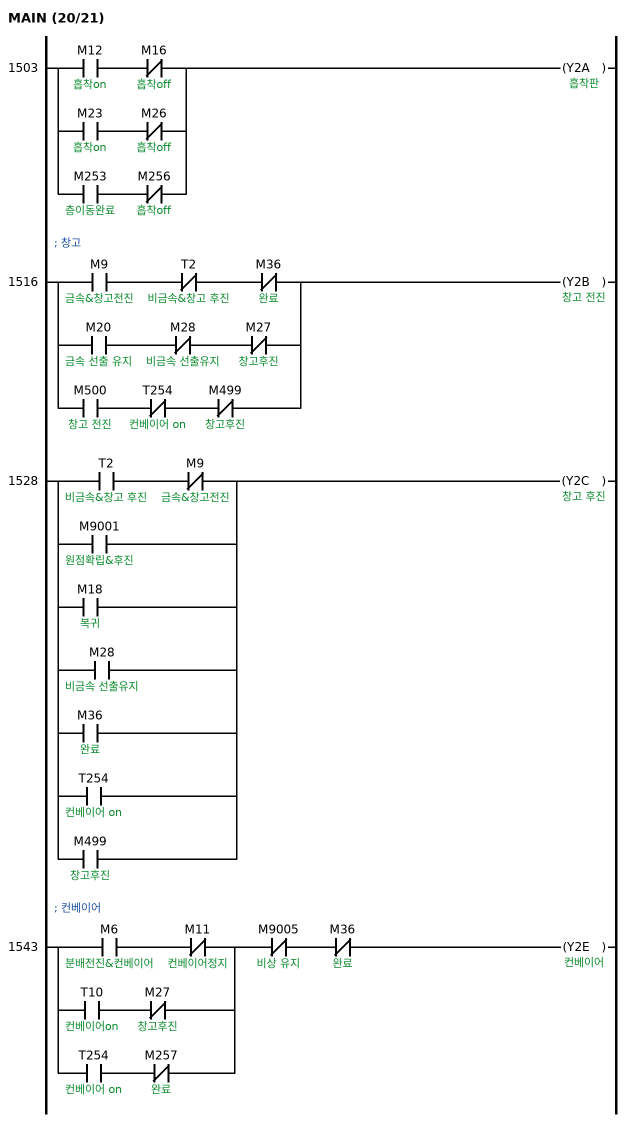
1503  LD      M12  ; 흡착on
      ANI     M16  ; 흡착off
      LD      M23  ; 흡착on
      ANI     M26  ; 흡착off
      ORB
      LD      M253  ; 층이동완료
      ANI     M256  ; 흡착off
      ORB
      OUT     Y2A  ; 흡착판
; 창고
1516  LD      M9  ; 금속&창고전진
      ANI     T2  ; 비금속&창고 후진
      ANI     M36  ; 완료
      LD      M20  ; 금속 선출 유지
      ANI     M28  ; 비금속 선출유지
      ANI     M27  ; 창고후진
      ORB
      LD      M500  ; 창고 전진
      ANI     T254  ; 컨베이어 on
      ANI     M499  ; 창고후진
      ORB
      OUT     Y2B  ; 창고 전진
1528  LD      T2  ; 비금속&창고 후진
      ANI     M9  ; 금속&창고전진
      OR      M9001  ; 원점확립&후진
      OR      M18  ; 복귀
      OR      M28  ; 비금속 선출유지
      OR      M36  ; 완료
      OR      T254  ; 컨베이어 on
      OR      M499  ; 창고후진
      OUT     Y2C  ; 창고 후진
; 컨베이어
1543  LD      M6  ; 분배전진&컨베이어
      ANI     M11  ; 컨베이어정지
      LD      T10  ; 컨베이어on
      ANI     M27  ; 창고후진
      ORB
      LD      T254  ; 컨베이어 on
      ANI     M257  ; 완료
      ORB
      ANI     M9005  ; 비상 유지
      ANI     M36  ; 완료
      OUT     Y2E  ; 컨베이어
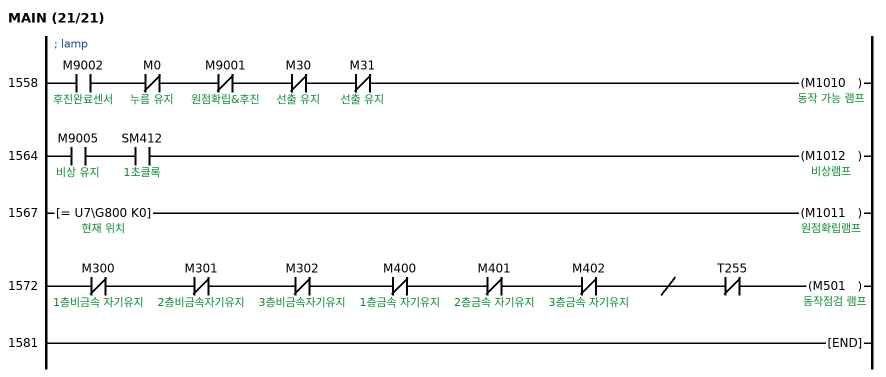
; lamp
1558  LD      M9002  ; 후진완료센서
      ANI     M0  ; 누름 유지
      ANI     M9001  ; 원점확립&후진
      ANI     M30  ; 선출 유지
      ANI     M31  ; 선출 유지
      OUT     M1010  ; 동작 가능 램프
1564  LD      M9005  ; 비상 유지
      AND     SM412  ; 1초클록
      OUT     M1012  ; 비상램프
1567  LD=     U7\G800 K0  ; 현재 위치
      OUT     M1011  ; 원점확립램프
1572  LDI     M300  ; 1층비금속 자기유지
      ANI     M301  ; 2층비금속자기유지
      ANI     M302  ; 3층비금속자기유지
      ANI     M400  ; 1층금속 자기유지
      ANI     M401  ; 2층금속 자기유지
      ANI     M402  ; 3층금속 자기유지
      INV
      ANI     T255
      OUT     M501  ; 동작점검 램프
1581  END
END_PROGRAM

// device comments not shown above
M13  ; 흡착 전진
M32  ; 흠
M37  ; 4개이상
T11  ; 리셋 타이머
T12  ; 리셋 타이머
D1014  ; 가공 횟수 지정
D1015  ; 가공 횟수
D1031  ; 1번선입
D1032  ; 2번선입
D1033  ; 3번 선입
D1034  ; 4번 선입
D1035  ; 5번 선입
D1036  ; 6번 선입
